// TIA Portal V19 export
DATA_BLOCK "HmiInterface"   // DB26
// stored: Access Published, MemoryReserve 100, Namespace Unit2.EM3
   VAR
      em : "LAF_typeEmInterface";
      jobs : "LAF_typeJobsInterface";
      sequence : "LAF_typeSequenceInterface";
      cm1SV112_Constraint1_Axis { S7_SetPoint := 'True'} : "LBC_typeAxisSimpleControlInterface_1";
      cm2SV113_Constraint2_Axis { S7_SetPoint := 'True'} : "LBC_typeAxisSimpleControlInterface_1";
      cm3SV115_Screw1_Axis { S7_SetPoint := 'True'} : "LEXCHANGETRAY_typeAxisSimpleControlInterface_2";
      cm4SV116_Screw2_Axis { S7_SetPoint := 'True'} : "LEXCHANGETRAY_typeAxisSimpleControlInterface_2";
      cm6SlideCylinder1 { S7_SetPoint := 'True'} : "LBC_Simple_typeTwoWayActuatorInterface";
      cm7hookClawCylinder1 { S7_SetPoint := 'True'} : "LBC_Simple_typeTwoWayActuatorInterface";
      cm8SlideCylinder2 { S7_SetPoint := 'True'} : "LBC_Simple_typeTwoWayActuatorInterface";
      cm9hookClawCylinder2 { S7_SetPoint := 'True'} : "LBC_Simple_typeTwoWayActuatorInterface";
      cm10SignalTM : "LEXCHANGETRAY_typeConstraintWorkstationIoSignalInterface";
      cm11PressureGaugeRs485 { S7_SetPoint := 'True'} : "typePressureGuageRs485Interface";
      em3Parameters { S7_SetPoint := 'True'} : "LAF_typeConstraintWorkstationEm3ParametersInterface";
   END_VAR
BEGIN
END_DATA_BLOCK
